Omron Sysmac Studio project Robotica_Data (Sysmac Studio 1.60.0.64010, StandardProject)

# Controller new_Controller_0: NX1P2-1040DT1 version 1.64
Task PrimaryTask (priority 4, period or condition 2000): Program0

VAR_GLOBAL RETAIN
    IN_POS1_VERDE AT %D100 : WORD;
    IN_POS1_AMARELO AT %D101 : WORD;
    IN_POS1_AZUL AT %D102 : WORD;
    IN_POS2_VERDE AT %D103 : WORD;
    IN_POS2_AMARELO AT %D104 : WORD;
    IN_POS2_AZUL AT %D105 : WORD;
    IN_POS3_VERDE AT %D106 : WORD;
    IN_POS3_AMARELO AT %D107 : WORD;
    IN_POS3_AZUL AT %D108 : WORD;
    RESET_DETECTION AT %D200 : BOOL;
    SYSTEM_READY AT %D201 : BOOL;
END_VAR
VAR_GLOBAL
    OUT_POS1_VERDE : BOOL;
    OUT_POS1_AMARELO : BOOL;
    OUT_POS1_AZUL : BOOL;
    OUT_POS2_VERDE : BOOL;
    OUT_POS2_AMARELO : BOOL;
    OUT_POS2_AZUL : BOOL;
    OUT_POS3_VERDE : BOOL;
    OUT_POS3_AMARELO : BOOL;
    OUT_POS3_AZUL : BOOL;
    OUTPUT_AMARELO_POS1 : BOOL;  (* at BuiltInIO://cpu/#0/Output_Bit_01 *)
    OUTPUT_AZUL_POS1 : BOOL;  (* at BuiltInIO://cpu/#0/Output_Bit_02 *)
    OUTPUT_VERDE_POS1 : BOOL;  (* at BuiltInIO://cpu/#0/Output_Bit_00 *)
    OUTPUT_AMARELO_POS2 : BOOL;  (* at BuiltInIO://cpu/#0/Output_Bit_04 *)
    OUTPUT_AZUL_POS2 : BOOL;  (* at BuiltInIO://cpu/#0/Output_Bit_05 *)
    OUTPUT_VERDE_POS2 : BOOL;  (* at BuiltInIO://cpu/#0/Output_Bit_03 *)
    OUTPUT_AMARELO_POS3 : BOOL;  (* at BuiltInIO://cpu/#0/Output_Bit_07 *)
    OUTPUT_AZUL_POS3 : BOOL;  (* at BuiltInIO://cpu/#0/Output_Bit_08 *)
    OUTPUT_VERDE_POS3 : BOOL;  (* at BuiltInIO://cpu/#0/Output_Bit_06 *)
END_VAR

PROGRAM Program0
VAR_EXTERNAL
    IN_POS1_VERDE : WORD;
    IN_POS1_AMARELO : WORD;
    IN_POS1_AZUL : WORD;
    IN_POS2_VERDE : WORD;
    IN_POS2_AMARELO : WORD;
    IN_POS2_AZUL : WORD;
    IN_POS3_VERDE : WORD;
    IN_POS3_AMARELO : WORD;
    IN_POS3_AZUL : WORD;
    OUTPUT_VERDE_POS1 : BOOL;
    OUTPUT_AMARELO_POS1 : BOOL;
    OUTPUT_AZUL_POS1 : BOOL;
    OUTPUT_VERDE_POS2 : BOOL;
    OUTPUT_AZUL_POS2 : BOOL;
    OUTPUT_VERDE_POS3 : BOOL;
    OUTPUT_AMARELO_POS3 : BOOL;
    OUTPUT_AZUL_POS3 : BOOL;
    RESET_DETECTION : BOOL;
    SYSTEM_READY : BOOL;
    OUTPUT_AMARELO_POS2 : BOOL;
END_VAR

(* Section Section0: ladder, written here as Structured Text *)

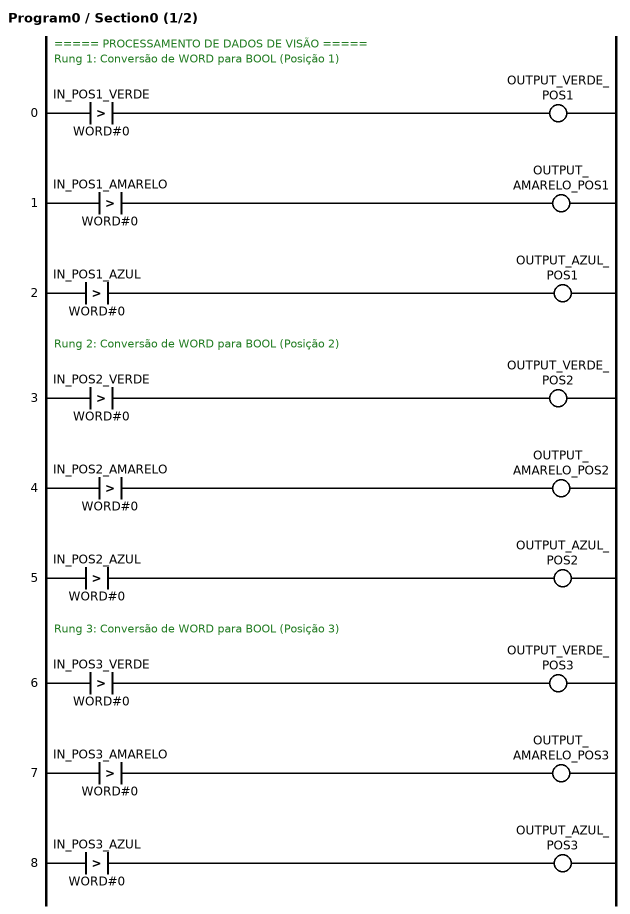
(* Rung 0: ===== PROCESSAMENTO DE DADOS DE VISÃO ===== / Rung 1: Conversão de WORD para BOOL (Posição 1) *)
OUTPUT_VERDE_POS1 := IN_POS1_VERDE > WORD#0;
(* Rung 1 *)
OUTPUT_AMARELO_POS1 := IN_POS1_AMARELO > WORD#0;
(* Rung 2 *)
OUTPUT_AZUL_POS1 := IN_POS1_AZUL > WORD#0;
(* Rung 3: Rung 2: Conversão de WORD para BOOL (Posição 2) *)
OUTPUT_VERDE_POS2 := IN_POS2_VERDE > WORD#0;
(* Rung 4 *)
OUTPUT_AMARELO_POS2 := IN_POS2_AMARELO > WORD#0;
(* Rung 5 *)
OUTPUT_AZUL_POS2 := IN_POS2_AZUL > WORD#0;
(* Rung 6: Rung 3: Conversão de WORD para BOOL (Posição 3) *)
OUTPUT_VERDE_POS3 := IN_POS3_VERDE > WORD#0;
(* Rung 7 *)
OUTPUT_AMARELO_POS3 := IN_POS3_AMARELO > WORD#0;
(* Rung 8 *)
OUTPUT_AZUL_POS3 := IN_POS3_AZUL > WORD#0;

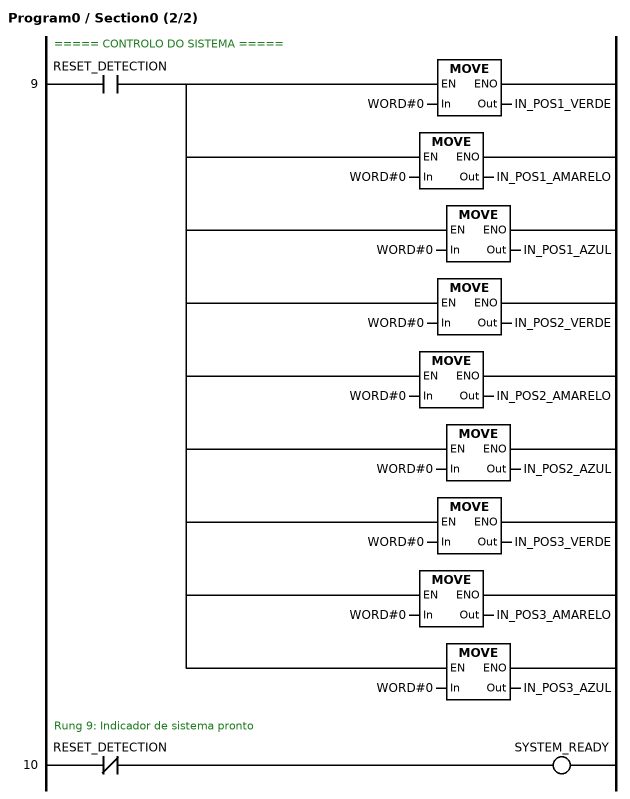
(* Rung 9: ===== CONTROLO DO SISTEMA ===== *)
IF RESET_DETECTION THEN
    IN_POS1_VERDE := WORD#0;
    IN_POS1_AMARELO := WORD#0;
    IN_POS1_AZUL := WORD#0;
    IN_POS2_VERDE := WORD#0;
    IN_POS2_AMARELO := WORD#0;
    IN_POS2_AZUL := WORD#0;
    IN_POS3_VERDE := WORD#0;
    IN_POS3_AMARELO := WORD#0;
    IN_POS3_AZUL := WORD#0;
END_IF;
(* Rung 10: Rung 9: Indicador de sistema pronto *)
SYSTEM_READY := NOT RESET_DETECTION;
END_PROGRAM